Staubli VAL3: clear.pgx

public program clear(num pX, num pY)
  local num i
  local num lLen
begin
  //---------------------------------
  //      C L E A R   L I N E
  //---------------------------------
  // Erase a pY line from the column
  // pX to end
  //
  //
  call typeLen(pX,pY," ",40-pX)
  gotoxy(pX,pY)
end
